// TIA Portal V19 export
TYPE "C701_VAR_IF_VEKR_TYPIC"
   STRUCT
      STO { ExternalAccessible := 'False'; ExternalVisible := 'False'; ExternalWritable := 'False'} : Struct   // Opsomming van alle storingen
         A001 : Bool;   // Storing van de motorbeveiliging van de pomp
         A002 : Bool;   // Fout temperatuurmeting vertrek
         A003 : Bool;   // Fout temperatuurmeting retour
         A004 : Bool;   // Fout drukmeting
         M001 : Bool;   // De motor is afgekoppeld via de werkschakelaar
      END_STRUCT;
   END_STRUCT;
END_TYPE
